Fanuc KAREL source: kt00096.KL

-- PROVISIONAL review KL for V1013-1; original PC SHA256 91c945a307e5b98f6c578eecc7539b7118d5b0a7d53e72c161397df46bd50d70
-- Incomplete behavior may be omitted. Consult companion uncertainty JSON. Do not deploy.
PROGRAM KT00096
%NOLOCKGROUP
VAR
  OUT : REAL
-- UNRESOLVED_DECL H1 type=002017
-- UNRESOLVED_DECL H2 type=002017
BEGIN
  -- UNRESOLVED_PC offsets 5-19; opcodes 2E,22,9D,33,B4
  -- UNRESOLVED_PC offsets 24-38; opcodes 2E,22,9D,33,B4
  -- UNRESOLVED_PC offsets 43-57; opcodes 2E,22,9D,33,B4
  -- UNRESOLVED_PC offsets 62-76; opcodes 2E,22,9D,33,B4
  -- UNRESOLVED_PC offsets 81-107; opcodes 22,9D,33,B3,22,9D,33,B3,54,64,23
  -- UNRESOLVED_PC offsets 112-116; opcodes 7F
END KT00096
